TYPE ST_RunEvent :
STRUCT
    dtTimestamp : DT; // Timestamp of the event (e.g., start, end)
    sEvent      : STRING(50); // Description of the event (e.g., "Started", "Completed")
END_STRUCT
END_TYPE

(* stored: Version 1.1.0.1, ProductVersion 3.1.4024.12
   DUT ST_RunEvent: Id {463b2fc5-9255-4504-ba3f-350c0399df15} *)
